PROGRAM MAIN

VAR_INPUT
	btnEstop		AT %I* : BOOL;
	btnStart		AT %I* : BOOL;
	btnStop			AT %I* : BOOL;
	btnReset		AT %I* : BOOL;
	btn_Reset		: BOOL;
	btnSoftEstop	: BOOL;
	btnTorchClean	: BOOL;
	Kuka_Ready		: BOOL;
	LogText			: STRING;
	BTN_LOG			: BOOL;
	Reset_State	: BOOL;
END_VAR

VAR
	fb_TimeStamp	: FB_UpdateTimeStamp;
	ModbusOn	: TON;
	ModbusOff	: TON;
	bOn			: BOOL;
	bLastOn		: BOOL;
END_VAR

	// =============================== Estop
		IF NOT btnEStop OR btnSoftEstop THEN
			ESTOP(); 
		END_IF
		
	// =============================== Reset
		IF btn_Reset THEN
			Reset_State := TRUE; 
		END_IF	
		
		IF btnReset THEN
			Reset_State := TRUE;
			IF NOT Reset_State THEN
				LOGFILE( sLogEvent	 := MSG.EVENT_BTN,
						sLogComp	 := MSG.COMP_OP_BTN, 
						sLogAction	 := MSG.ACTION_RESET, 
						 logFlag	 := TRUE);
			END_IF
		END_IF
			
		IF Reset_State THEN
			RESET_SEQ();
		END_IF
		
	// =============================== Kuka Ready	
		IF KR1.KROnline AND KR2.KROnline AND KR3.KROnline AND KR4.KROnline AND KR5.KROnline THEN
				MAIN.Kuka_Ready := TRUE;
		ELSE
				MAIN.Kuka_Ready := FALSE;	
		END_IF
		
	// =============================== Programme	
	fb_TimeStamp();
	IF fb_TimeStamp.timeValid THEN
			KUKA_IO();
			INFEED_RACK();
			COOL_RACK();
			JIG();
			AUTO_MODE();
			SAFETY_SENSOR();
			TL();
			
			//======================================= Modbus
			//Off time
			ModbusOn(IN:= NOT ModbusOff.Q, PT:= T#1S, Q=> bOn , ET=> );
			//On time
			ModbusOff(IN:= bOn, PT:= T#1S, Q=> , ET=> );
				
			IF bOn <> bLastOn THEN
				IF bON THEN
					COOL_RACK.bstart_Read := INFEED_RACK.bstart_Read := TRUE;
				ELSE
					COOL_RACK.bstart_Read := INFEED_RACK.bstart_Read := FALSE;
				END_IF
			END_IF
			bLastOn := bOn;
			// ================================================
		
			// ======================================= Torch Clean
			IF btnTorchClean THEN 
				TORCHCLEAN(); 
			ELSE 
				TORCHCLEAN.process_A:=0; 
			END_IF
		
			// ======================================= Operator Button
			IF btnStart THEN
				IF NOT AUTO_MODE.AutoMode THEN
					AUTO_MODE.Halt_Production := FALSE;
					LOGFILE( sLogEvent	 := MSG.EVENT_BTN,
							 sLogComp	 := MSG.COMP_OP_BTN, 
							 sLogAction	 := MSG.ACTION_START, 
							 logFlag	 := TRUE);
					AUTO_MODE.AutoMode := TRUE; 
					AUTO_MODE.Start_time := MAIN.fb_TimeStamp.SystemTime;
				ELSE
					AUTO_MODE.Halt_Production := FALSE;
					AUTO_MODE.AutoMode := TRUE; 
				END_IF
			END_IF
			
			IF btnStop THEN
				IF NOT AUTO_MODE.Halt_Production THEN
					LOGFILE( sLogEvent	 := MSG.EVENT_BTN,
							 sLogComp	 := MSG.COMP_OP_BTN, 
							 sLogAction	 := MSG.ACTION_STOP, 
							 logFlag	 := TRUE);
					KR1.bOutBit[1,0]:= FALSE;
					KR2.bOutBit[1,0]:= FALSE;
					KR3.bOutBit[1,0]:= FALSE;
					KR4.bOutBit[1,0]:= FALSE;
					KR5.bOutBit[1,0]:= FALSE;
					AUTO_MODE.Halt_Production := TRUE;
					AUTO_MODE.AutoMode := FALSE;
					Reset_State := FALSE;
				ELSE
					KR1.bOutBit[1,0]:= FALSE;
					KR2.bOutBit[1,0]:= FALSE;
					KR3.bOutBit[1,0]:= FALSE;
					KR4.bOutBit[1,0]:= FALSE;
					KR5.bOutBit[1,0]:= FALSE;
					AUTO_MODE.Halt_Production := TRUE;
					AUTO_MODE.AutoMode := FALSE;
					Reset_State := FALSE;
				END_IF
			END_IF
	END_IF

END_PROGRAM

(* stored: Version 1.1.0.1, ProductVersion 3.1.4024.12
   POU MAIN: Id {2e5786d8-6d11-41e5-a2a9-962bd5c7bdd1}, SpecialFunc None *)
